PROGRAM Axis05_Interlock
VAR
	Always_ON	:	BOOL	:=TRUE	;//상시 ON 
	Always_OFF	:	BOOL	:=FALSE	;//상시 OFF
END_VAR

// NETWORK 1

END_PROGRAM

(* stored: Version 1.1.0.1, ProductVersion 3.1.4024.15
   POU Axis05_Interlock: Id {baa90fa8-6f44-44e8-8b25-6afdea8e539e}, SpecialFunc None *)
